// TIA Portal V16 export
// export: Created 2024-02-03T21:03:33.1990585Z, ExportSetting WithDefaults, DisplayName Totally Integrated Automation Portal, DisplayVersion V16 Update 6, DisplayName TIA Portal Version Control Interface, DisplayVersion V16 Update 2, DisplayName TIA Portal Openness, DisplayVersion V16 Update 6, DisplayName SINAMICS Startdrive Advanced, DisplayVersion V16 Update 5, DisplayName SINAMICS Startdrive G130, G150, S120, S150, SINAMICS MV, S210, DisplayVersion V16 Update 5, DisplayName SINAMICS Startdrive G110M, G120, G120C, G120D, G120P, G115D, DisplayVersion V16 Update 5, DisplayName STEP 7 Professional, DisplayVersion V16 Update 6, DisplayName STEP 7 Safety, DisplayVersion V16, DisplayName WinCC Professional, DisplayVersion V16 Update 6
FUNCTION_BLOCK "test_blocks"   // FB2, LAD
{ S7_Optimized_Access := 'TRUE' }
VERSION : 0.1
// stored: AutoNumber true, IsIECCheckEnabled false, IsRetainMemResEnabled false, MemoryReserve 100, SetENOAutomatically false, UDAEnableTagReadback false
   VAR
      MC_POWER_Instance { S7_SetPoint := 'True'} : MC_POWER;
      MC_RESET_Instance { S7_SetPoint := 'True'} : MC_RESET;
      MC_HOME_Instance { S7_SetPoint := 'True'} : MC_HOME;
   END_VAR
BEGIN

REGION Network 1: Enable
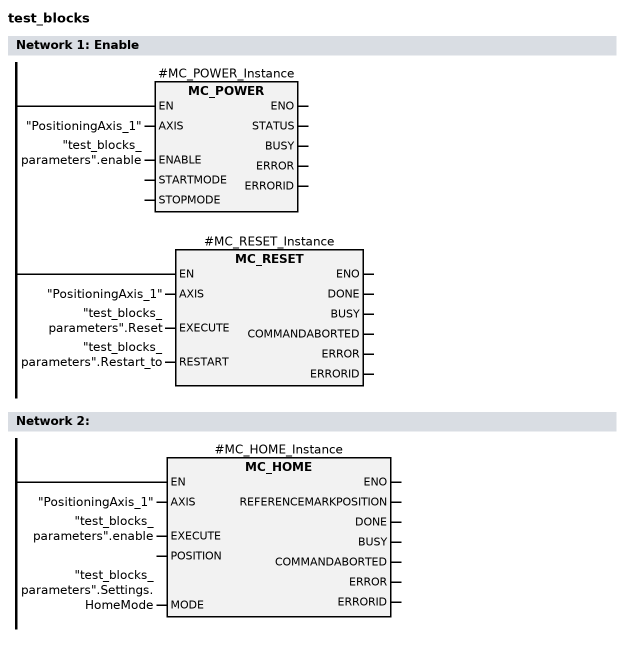
   RUNG wire#powerrail
      #MC_POWER_Instance.MC_POWER(Axis := "PositioningAxis_1", Enable := "test_blocks_parameters".enable, StartMode :=, StopMode :=, Status =>, Busy =>, Error =>, ErrorId =>)
   END_RUNG
   RUNG wire#powerrail
      #MC_RESET_Instance.MC_RESET(Axis := "PositioningAxis_1", Execute := "test_blocks_parameters".Reset, Restart := "test_blocks_parameters".Restart_to, Done =>, Busy =>, CommandAborted =>, Error =>, ErrorId =>)
   END_RUNG
   // the same network as SCL:
   #MC_POWER_Instance(Axis := "PositioningAxis_1", Enable := "test_blocks_parameters".enable);   // MC_POWER
   #MC_RESET_Instance(Axis := "PositioningAxis_1",   // MC_RESET
                      Execute := "test_blocks_parameters".Reset,
                      Restart := "test_blocks_parameters".Restart_to);
END_REGION

REGION Network 2
   RUNG wire#powerrail
      #MC_HOME_Instance.MC_HOME(Axis := "PositioningAxis_1", Execute := "test_blocks_parameters".enable, Position :=, Mode := "test_blocks_parameters".Settings.HomeMode, ReferenceMarkPosition =>, Done =>, Busy =>, CommandAborted =>, Error =>, ErrorId =>)
   END_RUNG
   // the same network as SCL:
   #MC_HOME_Instance(Axis := "PositioningAxis_1",   // MC_HOME
                     Execute := "test_blocks_parameters".enable,
                     Mode := "test_blocks_parameters".Settings.HomeMode);
END_REGION
END_FUNCTION_BLOCK
